RoboDK station: Part_on_conveyor.rdk

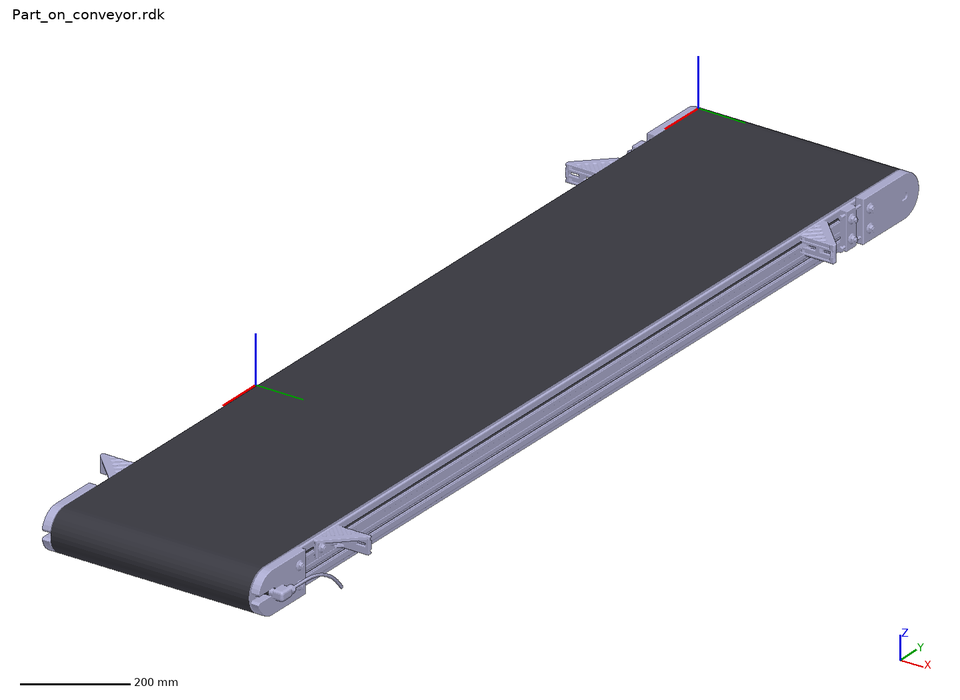
[picture v0: the station drawn from its stored meshes, robots at their saved joint values, targets as dots, program paths as lines]
Station Part_on_conveyor (saved by RoboDK 5.2.2). Poses are relative to the parent item; angles as X-Y-Z fixed-axis rotations.
  - frame Frame 1 at (0, 0, 0) mm
    - frame Conveyor Belt Base at (-430, -550, 210) mm, rotated rx 0 ry 0 rz -90 deg
      - robot Conveyor Belt: 1 axes
          modified DH rows (alpha deg, a mm, theta deg, d mm): 0, 0, 0, 0 linear
          base shift (0, 0, 0) mm, rotated rx 0 ry 90 rz 0 deg
          joint limits [-500000] to [500000]; home [0]; saved at [0]
        - frame Conveyor Box at (0, 0, 0) mm
      - frame New_Box 24X16 at (1400, 0, 0) mm
        - object BoxRef_24X16 at (0, 420, 0) mm, rotated rx 0 ry 0 rz -90 deg, size 398.1 x 610.2 x 267.5 mm, geometry from Box 24x16 closed.step
  - Python program Empty_Conveyor (listed below)
  - Python program New_Box (listed below)
  - Python program Conv_Move (listed below)
  - Python program Conv_Init_Position (listed below)
  - program Add_Box (3 instructions, listed below)
  - program Init (2 instructions, listed below)
  - program Main (4 instructions, listed below)

--- Python program Empty_Conveyor ---
# Type help("robolink") or help("robodk") for more information
# Press F5 to run the script
# Documentation: https://robodk.com/doc/en/RoboDK-API.html
# Reference:     https://robodk.com/doc/en/PythonAPI/index.html
# Note: It is not required to keep a copy of this file, your python script is saved with the station
from robolink import *    # RoboDK API
from robodk import *      # Robot toolbox
RDK = Robolink()

#----- CONSTANT -----
CONV_FRAME_NAME = 'Conveyor Box'

#----- PROGRAM -----
frame = RDK.Item(CONV_FRAME_NAME,ITEM_TYPE_FRAME)

if frame.Valid():
    for item in frame.Childs():
        if item.Type() == ITEM_TYPE_OBJECT:
            item.Delete()

--- Python program New_Box ---
# Type help("robolink") or help("robodk") for more information
# Press F5 to run the script
# Documentation: https://robodk.com/doc/en/RoboDK-API.html
# Reference:     https://robodk.com/doc/en/PythonAPI/index.html
# Note: It is not required to keep a copy of this file, your python script is saved with the station
from robolink import *    # RoboDK API
from robodk import *      # Robot toolbox
RDK = Robolink()



#----- Constante -----

REFERENCE_FRAME = 'Conveyor Box' # where the box will be moved
REFERENCE_FRAME_REF = 'New_Box 24X16' # ref for box

NEW_REF_OBJECT_NAME = 'BoxRef_24X16'
NEW_OBJECT_NAME = 'Box_24X16_On_Conveyor'



#------- Program ------
frame = RDK.Item(REFERENCE_FRAME, ITEM_TYPE_FRAME)
frame_ref = RDK.Item(REFERENCE_FRAME_REF, ITEM_TYPE_FRAME)

ref_obj = RDK.Item(NEW_REF_OBJECT_NAME, ITEM_TYPE_OBJECT)

RDK.Render(False)
if frame.Valid() and  ref_obj.Valid():
    ref_obj.Copy()
    new_obj = RDK.Paste()
    new_obj.setVisible(False)
    new_obj.setName(NEW_OBJECT_NAME)
    new_obj.setParent(frame_ref)
    RDK.Update()
    new_obj.setParentStatic(frame)
    new_obj.setVisible(True)
RDK.Render(True)

--- Python program Conv_Move ---
# Type help("robolink") or help("robodk") for more information
# Press F5 to run the script
# Documentation: https://robodk.com/doc/en/RoboDK-API.html
# Reference:     https://robodk.com/doc/en/PythonAPI/index.html
# Note: It is not required to keep a copy of this file, your python script is saved with the station
from robolink import *    # RoboDK API
from robodk import *      # Robot toolbox
RDK = Robolink()

#------ CONSTANT ------
MECHANISM_NAME = 'Conveyor Belt'
PART_TRAVEL_MM = -660

mechanism = RDK.Item(MECHANISM_NAME,itemtype=ITEM_TYPE_ROBOT)

if mechanism.Valid():
    mechanism.MoveJ(mechanism.Joints() + PART_TRAVEL_MM)

--- Python program Conv_Init_Position ---
# Type help("robolink") or help("robodk") for more information
# Press F5 to run the script
# Documentation: https://robodk.com/doc/en/RoboDK-API.html
# Reference:     https://robodk.com/doc/en/PythonAPI/index.html
# Note: It is not required to keep a copy of this file, your python script is saved with the station
from robolink import *    # RoboDK API
from robodk import *      # Robot toolbox
RDK = Robolink()

MECHANISM_NAME = 'Conveyor Belt'
mechanism = RDK.Item(MECHANISM_NAME,itemtype=ITEM_TYPE_ROBOT)

if mechanism.Valid():
    mechanism.setJoints([0])

--- program Add_Box (robot Conveyor Belt) ---
  Call New_Box
  Call Conv_Move
  Pause 5000 ms

--- program Init (robot Conveyor Belt) ---
  Call Conv_Init_Position
  Call Empty_Conveyor

--- program Main (robot Conveyor Belt) ---
  Call Init
  i=0
WHILE i<6
i=i+1
  Call Add_Box
  END
